Fanuc KAREL source: kx00024.KL

-- PROVISIONAL review KL for V770-1; original PC SHA256 a34c9d98136b32e6d03c9528c3f156f09274c4af3519d215714a4fcaf354ef5b
-- Incomplete behavior may be omitted. Consult companion uncertainty JSON. Do not deploy.
PROGRAM KX00024
%NOLOCKGROUP
VAR
  I : INTEGER
  J : INTEGER
  B : BOOLEAN
  F : FILE
  S : STRING[80]
-- UNRESOLVED_DECL P type=000102
-- UNRESOLVED_DECL CNF type=00001c
BEGIN
  -- UNRESOLVED_PC offsets 5-15; opcodes 9D,22,A5
  -- UNRESOLVED_PC offsets 20-35; opcodes 22,A4,23
  -- UNRESOLVED_PC offsets 40-44; opcodes 7F
END KX00024
